// TIA Portal V17 export
// export: Created 2025-03-07T09:17:44.6242598Z, ExportSetting WithDefaults, DisplayName Totally Integrated Automation Portal, DisplayVersion V17 Update 8, DisplayName TIA Portal Openness, DisplayVersion V17 Update 8, DisplayName TIA Portal Version Control Interface, DisplayVersion V17, DisplayName SINAMICS Startdrive Advanced, DisplayVersion V17 SP2, DisplayName SINAMICS Startdrive G110M, G120, G120C, G120D, G120P, G115D, DisplayVersion V17 SP2, DisplayName SINAMICS Startdrive G130, G150, S120, S150, SINAMICS MV, S210, DisplayVersion V17 SP2, DisplayName STEP 7 Professional, DisplayVersion V17 Update 8, DisplayName SINUMERIK ONE STEP 7 Toolbox, DisplayVersion V17 Update 12, DisplayName SINUMERIK 840D sl STEP 7 Toolbox, DisplayVersion V17 Update 12, DisplayName STEP 7 Safety, DisplayVersion V17 Update 6, DisplayName WinCC Advanced, DisplayVersion V17 Update 8
DATA_BLOCK "DB2011_MODES_GENERAL_MG2"   // DB2011
{ S7_Optimized_Access := 'FALSE'; DB_Accessible_From_OPC_UA := 'FALSE' }
AUTHOR : ETXETAR
VERSION : 1.0
// stored: AutoNumber false, DBAccessibleFromOPCUA false, DBAccessibleFromWebserver true, IsOnlyStoredInLoadMemory false, IsWriteProtectedInAS false
   VAR RETAIN
      GENERAL : "AUTO_SINGLE_SEMI_MANUAL";
      STEP_BY_STEP { S7_SetPoint := 'True'} : "MODES";
      MDA { S7_SetPoint := 'True'} : "MODES";
      REFERENCE { S7_SetPoint := 'True'} : "MODES";
      INCREMENTAL { S7_SetPoint := 'True'} : "INCREMENTAL";
      BA { S7_SetPoint := 'True'} : "BA_MODE";
   END_VAR
BEGIN
   // STEP_BY_STEP.MODE_SELECTED : STEP BY STEP MODE SELECTED
   // MDA.MODE_SELECTED : MDA MODE SELECTED
   // REFERENCE.MODE_SELECTED : REFERENCE MODE SELECTED
END_DATA_BLOCK
